Fanuc KAREL source: inv_ref.kl

PROGRAM INV_REF

VAR
	I : INTEGER
BEGIN
	I = 1
	WRITE('I = ', I, CR)
END INV_REF
